Staubli VAL3: READTRSF.pgx

public program readTrsf(num nHndl_, string x_sCol, num x_nRow, trsf& trPos_[], bool& x_bResult[])
  local bool l_bIsOK
  local num l_nColAsciiCode
  local bool l_bResult
begin
  // read X coordinate from spreadsheet
  call readNumValue(nHndl_,x_sCol,x_nRow,trPos_.x,x_bResult)
  if x_bResult
    // increment column number
    call _incrementCol(x_sCol,l_bIsOK)
    if l_bIsOK
      // read Y coordinate from spreadsheet
      call readNumValue(nHndl_,x_sCol,x_nRow,trPos_.y,x_bResult)
      if x_bResult
        // increment column number
        call _incrementCol(x_sCol,l_bIsOK)
        if l_bIsOK
          // read RZ coordinate from spreadsheet
          call readNumValue(nHndl_,x_sCol,x_nRow,trPos_.rz,x_bResult)
        endIf
      endIf
    endIf
  endIf
end
